(* PLC project range_sensor, Dassault Systèmes ControlBuild 2024x *)
(* stored: creationDateTime 2023-10-03T11:12:51-01:00 *)

(* This module simulates the behaviour of an over threshold sensor with a detection area. *)
FUNCTION_BLOCK equipment_library.range_sensor
  VAR_INPUT
    level : REAL := 0.0;
    sensorSupply : BOOL := true;
  END_VAR
  VAR_OUTPUT
    rangeSensor : BOOL := false;
  END_VAR
  VAR CONSTANT
    threshold : REAL := 500.0;
    range : REAL := 10.0;
    wiringLogic : BOOL := true;
  END_VAR
  VAR
    d_sensor : BOOL := false;
    v_d_sensor : BOOL := false;
  END_VAR


ACTION C_source_code:
/* ----------------------------------------------------------------	*/
/* Type : Model of Operative Behaviour					*/
/* Category :  Sensors							*/
/* Author : Dassault Systemes						*/
/* Update date : June 2018							*/
/* ----------------------------------------------------------------	*/
/* This module simulates the behaviour 					*/
/* of an over threshold sensor with a detection area.			*/
/* ----------------------------------------------------------------	*/
/* In the case of a faulty element, it takes the fault value else 	*/
/* it takes the state of the sensor in function of its wiring logic.	*/ 
/* ----------------------------------------------------------------	*/

if (d_sensor) rangeSensor = v_d_sensor;
else
	if ( sensorSupply ) rangeSensor = ((level >= threshold) & (level <= (threshold + range))) ^ ! wiringLogic;
	else rangeSensor = 0;
END_ACTION
END_FUNCTION_BLOCK
